INTERFACE ITestBase_t

METHOD PUBLIC FINAL _cleanup : ERetCode_t
VAR_INPUT
END_VAR
END_METHOD

METHOD PUBLIC FINAL _execute : ERetCode_t
VAR_INPUT
END_VAR
END_METHOD

METHOD PUBLIC FINAL _prepare : ERetCode_t
VAR_INPUT
END_VAR
END_METHOD

METHOD getClassname : ObjectId_t
VAR_INPUT
END_VAR
END_METHOD

METHOD getId : ObjectId_t
VAR_INPUT
END_VAR
END_METHOD

METHOD getMessage : StrMessage_t
VAR_INPUT
END_VAR
END_METHOD

METHOD getPath : ObjectId_t
VAR_INPUT
END_VAR
END_METHOD

PROPERTY Result : STestcase_t
GET
END_GET
END_PROPERTY

END_INTERFACE

(* stored: Version 1.1.0.1, ProductVersion 3.1.4024.12
   Itf ITestBase_t: Id {9c48b1f4-ee79-43bd-b9a3-d78583bb60da}
   Method _cleanup: Id {fafc9c7e-f319-4379-b168-0ec8f0292d03}
   Method _execute: Id {acf175e3-b737-4368-87ef-537fb8e7d94a}
   Method _prepare: Id {2a2e458a-0f88-4594-94f6-e3fb93469a62}
   Method getClassname: Id {80fac9dc-a047-463f-aced-f02760d617fc}
   Method getId: Id {0f51fb20-4fae-474a-bdd3-960651b92a0f}
   Method getMessage: Id {61957595-151b-4032-8e9c-f69bc6b8620a}
   Method getPath: Id {826500ad-9e52-4726-a94b-08a67a71ffe5}
   Property Result: Id {1565c885-bd5b-4f76-bea6-bae078ea3d58}
   Get Get: Id {ec1bfcd2-1589-4bca-af07-92322c474187} *)
